// SIMATIC S7-200 project (STEP 7-Micro/WIN), CPU 224XP CN REL 02.01

SYMBOL_TABLE 用户定义1
传感器1             I0.0
传感器2             I0.1
传感器3             I0.2
传感器4             I0.3
传感器5             I0.4
传感器6             I0.5
传感器7             I0.6
传感器8             I0.7
启动1              M1.0
启动2              M2.0
启动3              M3.0
启动4              M4.0
启动5              M5.0
启动6              M6.0
启动7              M7.0
启动8              M8.0
停止1              M1.1
停止2              M2.1
停止3              M3.1
停止4              M4.1
停止5              M5.1
停止6              M6.1
停止7              M7.1
停止8              M8.1
暂停1              M1.2
暂停2              M2.2
暂停3              M3.2
暂停4              M4.2
暂停5              M5.2
暂停6              M6.2
暂停7              M7.2
暂停8              M8.2
堵袋1              M1.3
堵袋2              M2.3
堵袋3              M3.3
堵袋4              M4.3
堵袋5              M5.3
堵袋6              M6.3
堵袋7              M7.3
堵袋8              M8.3
END_SYMBOL_TABLE

ORGANIZATION_BLOCK 主程序:OB1
TITLE=程序注释
BEGIN
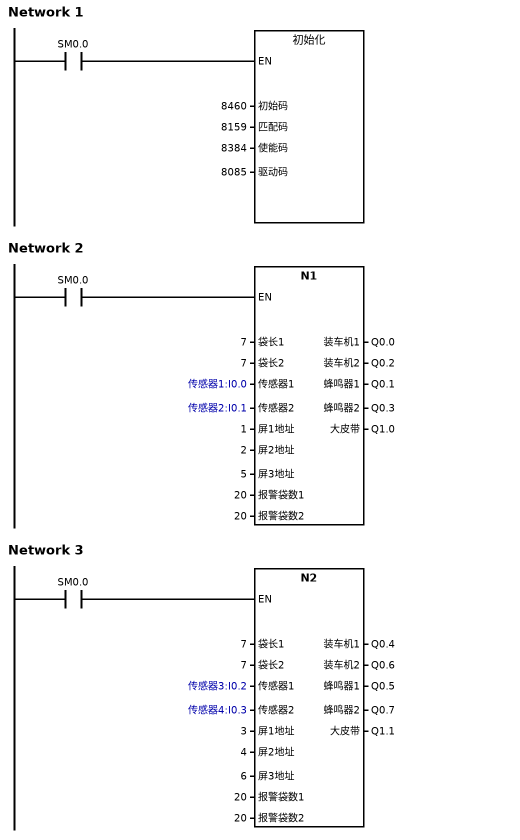
Network 1
LD     SM0.0
CALL   初始化:SBR0, 8460, 8159, 8384, 8085
Network 2
LD     SM0.0
CALL   N1:SBR32, 7, 7, 传感器1:I0.0, 传感器2:I0.1, 1, 2, 5, 20, 20, Q0.0, Q0.2, Q0.1, Q0.3, Q1.0
Network 3
LD     SM0.0
CALL   N2:SBR1, 7, 7, 传感器3:I0.2, 传感器4:I0.3, 3, 4, 6, 20, 20, Q0.4, Q0.6, Q0.5, Q0.7, Q1.1
END_ORGANIZATION_BLOCK

// SBR0: protected block, not included

// SBR1: protected block, not included

// SBR32: protected block, not included

// INT0: protected block, not included
